ABB RobotStudio station: CycleTime_Simu.rspag

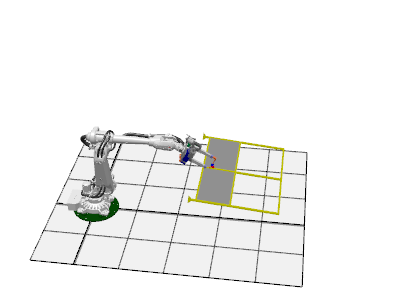
--- station ---
Station CycleTime_Simu (saved by RobotStudio 24.3.10835.0)
Controller IRB5720_90_300_LID, task T_ROB1: task frame (RAPID world) sits at (0, 0, 60) mm in the station
Controller IRB5720_90_300_LID
  mechanical unit ROB_1: IRB5720_90_300_MH6_01, 6 joints, base frame (0, 0, 0) mm
Layout (positions relative to the parent item):
  - IRB5720_90_300_MH6_01 [mechanism, from %ABB.RobotStudio.Models.IRB5720%\IRB5720_90_300_MH6_01.rslib] at (0, 0, 60) mm; joint values [0, 0, 0, 0, 0.5236, 0] (rad or m)
  - Robot BasePlate Type C_60 mm [part], size 1099.7 x 1099.7 x 60 mm
  - GWT_S1_0 [mechanism, from Tools\GWT_S1_0.rslib] at (2155.89, 0, 1883.5) mm, rotated rx 180 ry 60 rz 180 deg; joint values [0.1125] (rad or m)
  - Fence_2500 [graphiccomponentgroup, from Equipment\Fence_2500.rslib] at (2404.1, -992.56, 1301.23) mm, rotated rx 180 ry 84.5 rz 180 deg
    - Body 1 [part, from Equipment\Fence_2500.rslib]
    - Body 2 [part, from Equipment\Fence_2500.rslib]
  - RapidVariable [smart component, from Components\RapidVariable.rslib]
      properties: DataType=num; Controller=IRB5720_90_300_LID; Task=T_ROB1; Module=CycleTime; Variable=nTotalCycleTime; Value=12.396
  - MarkupControl [smart component, from Components\MarkupControl.rslib]
      properties: Markup=Markup_1; Text=12.396; Visible=true; Position=[2.941117 1.249541 1.252068]; BackColor=-4144960; ForeColor=-16777216; FontSize=32; Topmost=true
  - Timer [smart component, from Components\Timer.rslib]
      properties: StartTime=0; Interval=0.1; Repeat=true; CurrentTime=582.706
Attachment: GWT_S1_0 is attached to IRB5720_90_300_MH6_01 / Link6
Station logic (signal -> signal, property => property):
  Timer.Output -> RapidVariable.Get
  RapidVariable.Value => MarkupControl.Text
Targets, tools, work objects and paths stored in the station and not in the controller backup, written as RAPID:
! task T_ROB1
MODULE Toto
  PERS tooldata GWT_S1:=[TRUE,[[0,0,732.5],[0.707106781,0,-0.707106781,0]],[1,[0,0,100],[1,0,0,0],0,0,0]];
ENDMODULE


--- Controller Data/IRB5720_90_300_LID/RAPID/TASK1/PROGMOD/CycleTime.modx ---
MODULE CycleTime
    VAR clock cCycleTime;
    VAR num nCycleDone:=0;
    VAR num nSecondesPerCycle;
    VAR num nCyclePerHour;
    VAR num nCyclePerMinute;
    VAR num nTotalCycleTime:=0;
    VAR num nAverageSecondsPerCycle;
    VAR num nMinCycleTime:=9999999;
    VAR num nMaxCycleTime:=0;
    VAR num nLastCycleTime;

    PROC main()
        StartSimulation;
        FOR i FROM 1 TO 10 DO
            SimulateCycle;
            CycleComplete;
        ENDFOR
        PrintStatistics;
    ENDPROC

    PROC StartSimulation()
        TPErase;
        ClkStop cCycleTime;
        ClkReset cCycleTime;
        ClkStart cCycleTime;
    ENDPROC

    PROC CycleComplete()
        nLastCycleTime:=ClkRead(cCycleTime);
        ClkReset cCycleTime;
        ClkStart cCycleTime;
        Incr nCycleDone;
        nTotalCycleTime:=nTotalCycleTime+nLastCycleTime;
        UpdateStatistics;
    ENDPROC

    PROC PrintStatistics()
        TPWrite "Cycle Time Statistics:";
        TPWrite " Total Cycles Time: "\num:=nTotalCycleTime;
        TPWrite " Total Cycles: "\num:=nCycleDone;
        TPWrite " Average Cycle Time: "\num:=nAverageSecondsPerCycle;
        TPWrite " Min Cycle Time: "\num:=nMinCycleTime;
        TPWrite " Max Cycle Time: "\num:=nMaxCycleTime;
        TPWrite " Cycles per Hour: "\num:=nCyclePerHour;
        TPWrite " Cycles per Minute: "\num:=nCyclePerMinute;
    ENDPROC

    PROC SimulateCycle()
        WaitTime 1+((Rand()/32767)*0.5);
    ENDPROC

    PROC UpdateStatistics()
        IF (nLastCycleTime<nMinCycleTime) THEN
            nMinCycleTime:=nLastCycleTime;
        ENDIF
        IF (nLastCycleTime>nMaxCycleTime) THEN
            nMaxCycleTime:=nLastCycleTime;
        ENDIF
        nSecondesPerCycle:=nTotalCycleTime/nCycleDone;
        nCyclePerHour:=3600/nSecondesPerCycle;
        nCyclePerMinute:=60/nSecondesPerCycle;
        nAverageSecondsPerCycle:=nTotalCycleTime/nCycleDone;
    ENDPROC
ENDMODULE

--- Controller Data/IRB5720_90_300_LID/SYSPAR/EIO.cfg ---
EIO:CFG_1.0:7:0::
#
VIRTUAL_NETWORK:

      -Name "Virtual" -Label "Virtual Device Network"

#CTRL_SIGNATURE:he4/TkIMnw9nieK+ZICafPjETB/OQ5PMJRTCNxa4TD+PCQpCvghFiqirC5Y2wtgLDNYrxXZbmFo/4XPtA0bcsA==

--- Controller Data/IRB5720_90_300_LID/SYSPAR/PROC.cfg ---
PROC:CFG_1.0:7:0::

#CTRL_SIGNATURE:Dfzu9x1Ycvkd8lJYFuwW7gnrTbOTYkEJOiXphaxTue+Itf4eWjk9bu7hOCYXCSyQfUkNYkI1RRwwkOpyv1L9Bw==
